TYPE ST_EasyTempPara :
STRUCT
	bTuned : BOOL;
	stPID : ST_CTRL_ParaController;
	stPara: ST_CTRL_TempCtrlParameter;
END_STRUCT
END_TYPE

(* stored: Version 1.1.0.1, ProductVersion 3.1.4024.12
   DUT ST_EasyTempPara: Id {834ec6fb-f36c-40c9-8905-54b4a1ffeed0} *)
